// SIMATIC S7-200 project (STEP 7-Micro/WIN), CPU 221 REL 01.10

ORGANIZATION_BLOCK 主程序:OB1
TITLE=程序注释
BEGIN
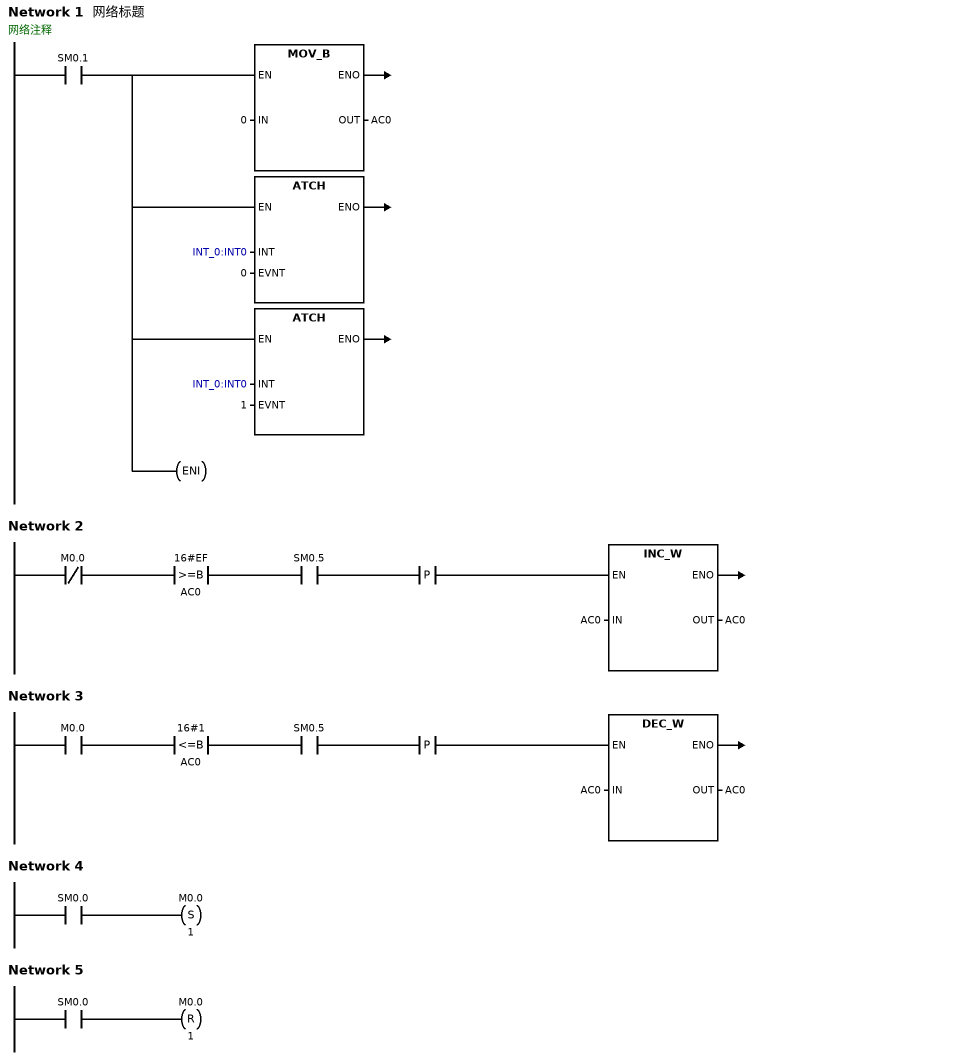
Network 1 // 网络标题
// 网络注释
LD     SM0.1
MOVB   0, AC0
ATCH   INT_0:INT0, 0
ATCH   INT_0:INT0, 1
ENI
Network 2
LDN    M0.0
AB>=   16#EF, AC0
A      SM0.5
EU
INCW   AC0
Network 3
LD     M0.0
AB<=   16#1, AC0
A      SM0.5
EU
DECW   AC0
Network 4
LD     SM0.0
S      M0.0, 1
Network 5
LD     SM0.0
R      M0.0, 1
END_ORGANIZATION_BLOCK
